(* LS Electric XG5000 project: XMC_ACDrive_FBs *)
(* sample programs for LS AC Drive function blocks. *)
(* PLC LSPLC *)
(* module base 0 slot 0: Input/Output Module:XMC-DN24 (DC 24V Input 8Points/TR output 16Points) *)
(* module base 0 slot 1: Internal Analog Input/Output:XMF-AH04E (A/D voltage/current 2 channels, D/A voltage 2 channels) *)
(* task Periodic Task: Kind=2 *)
(* task Initialization Task: Kind=1 *)
(* task NC Program: Kind=6 *)

PROGRAM ECAT_Connect_Example (* task: Scan Program *)
VAR
    Connect_Error : BOOL; (* status that LS_Connect has an error *)
    Connect_ErrorID : WORD; (* LS_Connect Error number *)
    Connect_INST : LS_CONNECT; (* LS_Connect fb *)
    Disconnect_Error : BOOL; (* status that LS_Disconnect has an error *)
    Disconnect_ErrorID : WORD; (* Error Number for LS_Disconnect FB *)
    Disconnect_INST : LS_DISCONNECT; (* LS_Disconnect fb *)
    Execute_Connect : BOOL; (* Execute LS_Connect fb *)
    Execute_Disconnect : BOOL; (* execute LS_Disconnect fb *)
END_VAR

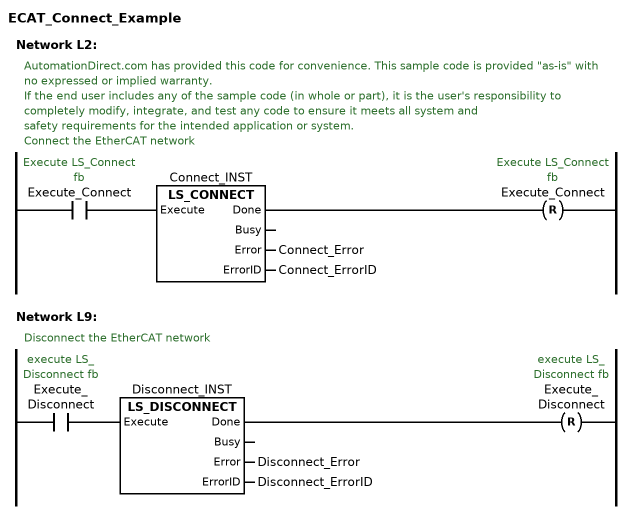
(* AutomationDirect.com has provided this code for convenience. This sample code is provided "as-is" with no expressed or implied warranty. / If the end user includes any of the sample code (in whole or part), it is the user's responsibility to completely modify, integrate, and test any code to ensure it meets all system and / safety requirements for the intended application or system. *)
(* Connect the EtherCAT network *)
(* Rung L2 *)
Connect_INST(Execute := Execute_Connect, Error => Connect_Error, ErrorID => Connect_ErrorID);
IF Connect_INST.Done THEN Execute_Connect := FALSE; END_IF;
(* Disconnect the EtherCAT network *)
(* Rung L9 *)
Disconnect_INST(Execute := Execute_Disconnect, Error => Disconnect_Error, ErrorID => Disconnect_ErrorID);
IF Disconnect_INST.Done THEN Execute_Disconnect := FALSE; END_IF;
END_PROGRAM

PROGRAM LS_InverterControl_Example (* task: Scan Program *)
(* example program for LS_InverterControl function block *)
VAR
    Axis1 : UINT; (* used to tell MC function blocks to use axis 1 *)
    EnableOP : BOOL;
    EnableRamp : BOOL;
    Execute_InverterControl : BOOL; (* execute the LS_InverterControl fb *)
    FaultReset : BOOL;
    Halt : BOOL;
    InveterControl_Error : BOOL; (* error status for LS_InverterControl *)
    InveterControl_ErrorID : WORD; (* error identification for LS_InverterControl *)
    InveterControl_INST : LS_INVERTERCONTROL; (* LS_InverterControl function block *)
    QuickStop : BOOL;
    ReferenceRamp : BOOL;
    SwitchOn : BOOL;
    UnlockRamp : BOOL;
    VoltageEn : BOOL;
END_VAR

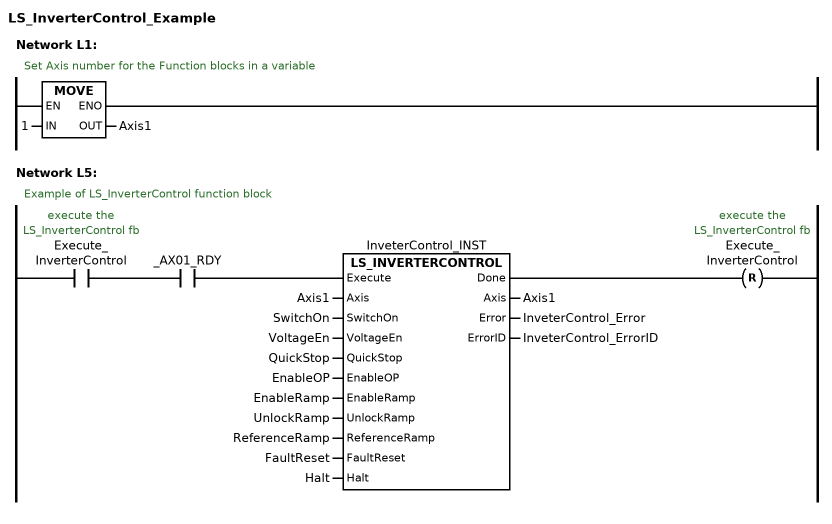
(* Set Axis number for the Function blocks in a variable *)
(* Rung L1 *)
Axis1 := 1;
(* Example of LS_InverterControl function block *)
(* Rung L5 *)
InveterControl_INST(Execute := Execute_InverterControl AND _AX01_RDY, Axis := Axis1, SwitchOn := SwitchOn, VoltageEn := VoltageEn, QuickStop := QuickStop, EnableOP := EnableOP, EnableRamp := EnableRamp, UnlockRamp := UnlockRamp, ReferenceRamp := ReferenceRamp, FaultReset := FaultReset, Halt := Halt, Axis => Axis1, Error => InveterControl_Error, ErrorID => InveterControl_ErrorID);
IF InveterControl_INST.Done THEN Execute_InverterControl := FALSE; END_IF;
END_PROGRAM

PROGRAM LS_InverterStatus_Example (* task: Scan Program *)
(* example program for LS_InverterStatus1 and LS_InverterStatus2 function blocks. *)
VAR
    Axis1 : UINT; (* used to tell MC function blocks to use axis 1 *)
    Execute_InverterStatus : BOOL; (* enable the LS_InverterStatus function blocks *)
    Fault : BOOL; (* fault status *)
    LimitActive : BOOL; (* limit active status *)
    OpEn : BOOL; (* Operation enabled status *)
    QuickStop : BOOL; (* Quick stop status *)
    Remote : BOOL; (* remote control status *)
    Status1_Enabled : BOOL; (* Enabled status for LS_InverterStatus1 *)
    Status1_Error : BOOL; (* error status for LS_InverterStatus1 *)
    Status1_ErrorID : WORD; (* error identification for LS_InverterStatus1 *)
    Status1_INST : LS_INVERTERSTATUS1; (* LS_InverterStatus1 function block *)
    Status1_RdySwitchOn : BOOL; (* Ready to switch on Status *)
    Status2_Enabled : BOOL; (* LS_InverterStatus2 enabled status *)
    Status2_Error : BOOL; (* error status for LS_InverterStatus2 *)
    Status2_ErrorID : WORD; (* error identification for LS_InverterStatus2 *)
    Status2_INST : LS_INVERTERSTATUS2; (* LS_InverterStatus2 function block *)
    SwitchedOn : BOOL; (* Switched on status *)
    SwOnDisable : BOOL; (* Switch on disabled status *)
    TargetReach : BOOL; (* target reached status *)
    VoltageEn : BOOL; (* Voltage Enabled status *)
    Warning : BOOL; (* warning status *)
END_VAR

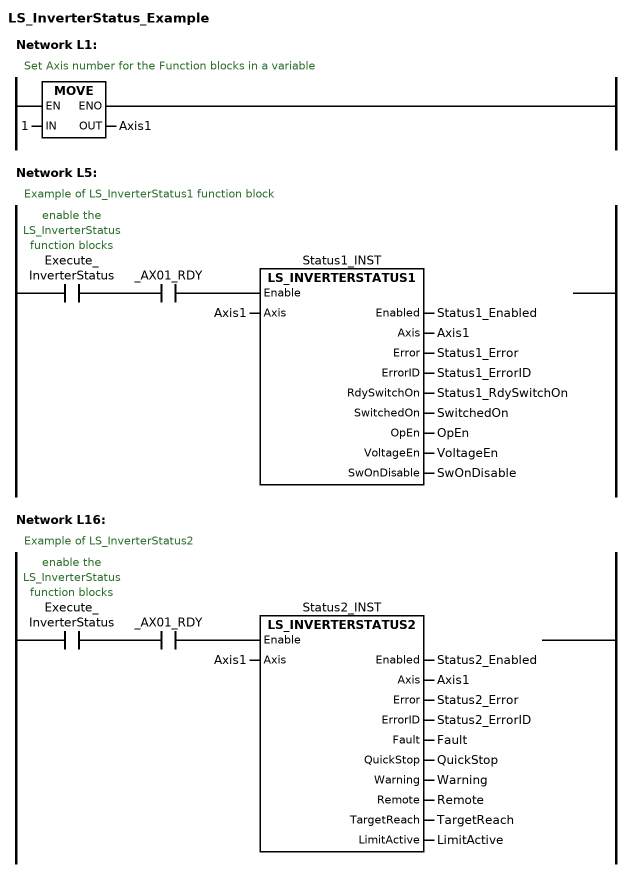
(* Set Axis number for the Function blocks in a variable *)
(* Rung L1 *)
Axis1 := 1;
(* Example of LS_InverterStatus1 function block *)
(* Rung L5 *)
Status1_INST(Enable := Execute_InverterStatus AND _AX01_RDY, Axis := Axis1, Enabled => Status1_Enabled, Axis => Axis1, Error => Status1_Error, ErrorID => Status1_ErrorID, RdySwitchOn => Status1_RdySwitchOn, SwitchedOn => SwitchedOn, OpEn => OpEn, VoltageEn => VoltageEn, SwOnDisable => SwOnDisable);
(* Example of LS_InverterStatus2 *)
(* Rung L16 *)
Status2_INST(Enable := Execute_InverterStatus AND _AX01_RDY, Axis := Axis1, Enabled => Status2_Enabled, Axis => Axis1, Error => Status2_Error, ErrorID => Status2_ErrorID, Fault => Fault, QuickStop => QuickStop, Warning => Warning, Remote => Remote, TargetReach => TargetReach, LimitActive => LimitActive);
END_PROGRAM

PROGRAM LS_InverterWriteVel_Example (* task: Scan Program *)
(* example program for LS_InverterWriteVel function block *)
VAR
    Axis1 : UINT; (* used to tell MC function blocks to use axis 1 *)
    Execute_WriteVelocity : BOOL; (* command to execute the LS_InverterWriteVel *)
    TargetVel : INT; (* target velocity in rpm *)
    WriteVelocity_Error : BOOL; (* error status for LS_InverterWriteVel *)
    WriteVelocity_ErrorID : WORD; (* error identification for LS_InverterWriteVel *)
    WriteVelocity_INST : LS_INVERTERWRITEVEL; (* LS_InverterWriteVel function block *)
END_VAR

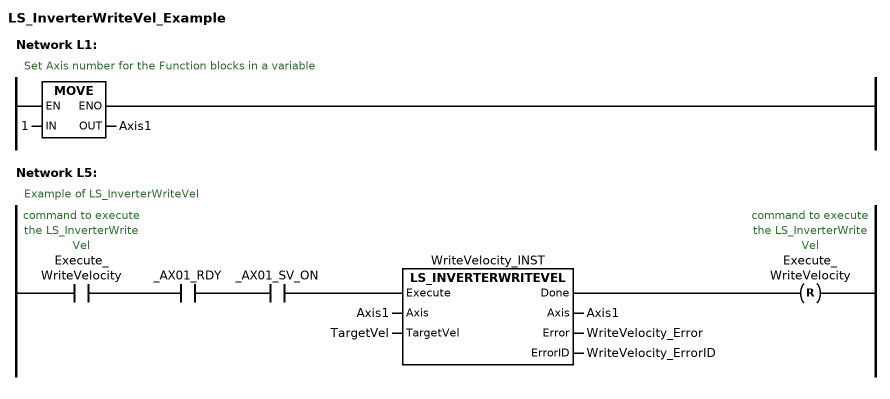
(* Set Axis number for the Function blocks in a variable *)
(* Rung L1 *)
Axis1 := 1;
(* Example of LS_InverterWriteVel *)
(* Rung L5 *)
WriteVelocity_INST(Execute := Execute_WriteVelocity AND _AX01_RDY AND _AX01_SV_ON, Axis := Axis1, TargetVel := TargetVel, Axis => Axis1, Error => WriteVelocity_Error, ErrorID => WriteVelocity_ErrorID);
IF WriteVelocity_INST.Done THEN Execute_WriteVelocity := FALSE; END_IF;
END_PROGRAM

PROGRAM LS_InverterReadVel_Example (* task: Scan Program *)
(* LS_InverterReadVel function block example program *)
VAR
    ActualVel : INT; (* actual velocity for AC drive *)
    Axis1 : UINT; (* used to tell MC function blocks to use axis 1 *)
    Execute_ReadVelocity : BOOL; (* execute the LS_InverterReadVel function block *)
    ReadVelocity_Enabled : BOOL; (* enabled status for LS_InverterReadVel *)
    ReadVelocity_Error : BOOL; (* error status for LS_InverterReadVel *)
    ReadVelocity_ErrorID : WORD; (* error identification for LS_InverterReadVel *)
    ReadVelocity_INST : LS_INVERTERREADVEL; (* LS_InverterReadVel function block *)
END_VAR

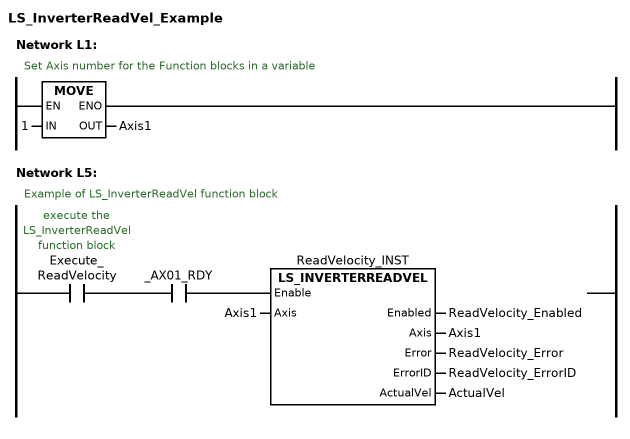
(* Set Axis number for the Function blocks in a variable *)
(* Rung L1 *)
Axis1 := 1;
(* Example of LS_InverterReadVel function block *)
(* Rung L5 *)
ReadVelocity_INST(Enable := Execute_ReadVelocity AND _AX01_RDY, Axis := Axis1, Enabled => ReadVelocity_Enabled, Axis => Axis1, Error => ReadVelocity_Error, ErrorID => ReadVelocity_ErrorID, ActualVel => ActualVel);
END_PROGRAM